FUNCTION_BLOCK STRUCT_MUX (* Service Interface Function Block Type *)
  (* Standard: 61499-2; Description: Copyright (c) This program and the accompanying materials are made available under the terms of the Eclipse Public License 2.0 which is available at https://www.eclipse.org/legal/epl-2.0/ SPDX-License-Identifier: EPL-2.0 *)
  {SET_ATTRIBUTE(GenericClassName, 'GEN_STRUCT_MUX')}
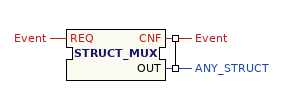
  EVENT_INPUT
    REQ; (* Normal Execution Request *)
  END_EVENT
  EVENT_OUTPUT
    CNF WITH OUT; (* Execution Confirmation *)
  END_EVENT
  VAR_OUTPUT
    OUT : ANY_STRUCT; (* Output *)
  END_VAR
  (* Service APPLICATION/RESOURCE: Service Interface Function Block Type *)
END_FUNCTION_BLOCK
